TYPE stCommand_Settings :
STRUCT
	Name : STRING;
	Velocity: LREAL;
	Acceleration: LREAL;
	Target: stTarget;
	Joints: stJoint6;
	Pose: ST_Pose;
	Pin: UINT;
	bValue: BOOL;
	fValue: REAL;
	nValue: INT;
	ID: UINT;
END_STRUCT
END_TYPE

(* stored: Version 1.1.0.1, ProductVersion 3.1.4026.18
   DUT stCommand_Settings: Id {8fac1be0-eb98-4b37-aae0-7d9ddbd25ee2} *)
